// Mitsubishi GX Works2 project: zadatak_1   PLC: FX3S

// task Task_01 (event TRUE, interval 0, priority 31): POU_01

PROGRAM POU_01
VAR
  system_on : BOOL;
  start : BOOL;
  stop_all : BOOL;
  start_all : BOOL;
  fsm_1 : fsm;
  pump_on : BOOL;
  goto_1 : BOOL;
  goto_2 : BOOL;
  goto_3 : BOOL;
  goto_4 : BOOL;
  goto_0 : BOOL;
  cur_state : INT;
  s_0 : BOOL;
  s_1 : BOOL;
  s_2 : BOOL;
  s_3 : BOOL;
  s_4 : BOOL;
  sensor_2 : BOOL;
END_VAR
VAR CONSTANT
  pause : TIME := T#10s;
END_VAR
VAR
  elapsed_time : TIME;
  sensor_1 : BOOL;
  water_rising : BOOL;
  valve_1 : BOOL;
  motor : BOOL;
  water_falling : BOOL;
  valve_2 : BOOL;
  alarm : BOOL;
  TON_1 : TON;
  cnt_cycles_1 : cnt_cycles;
  done : BOOL;
  blink_1 : blink;
  lamp : BOOL;
END_VAR
(* structured ladder/FBD written out as ST: instructions are called as NAME(EN, inputs, outputs); _pN, _eN, _tN stand for wires *)
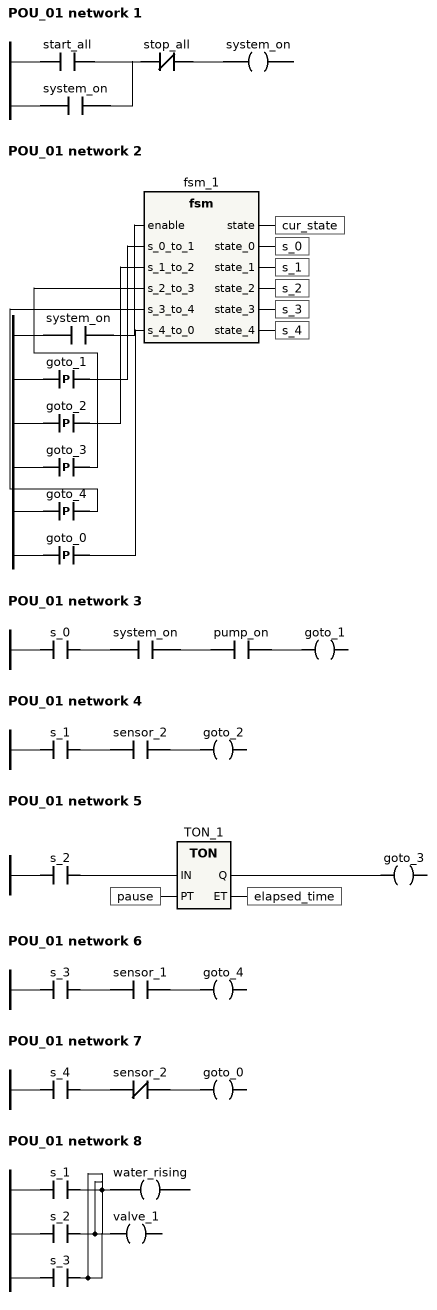
(* network 1 *)
system_on := (start_all OR system_on) AND NOT stop_all;
(* network 2 *)
fsm_1(enable := system_on, s_0_to_1 := LDP(TRUE, goto_1), s_1_to_2 := LDP(TRUE, goto_2), s_2_to_3 := LDP(TRUE, goto_3), s_3_to_4 := LDP(TRUE, goto_4), s_4_to_0 := LDP(TRUE, goto_0), state => cur_state, state_0 => s_0, state_1 => s_1, state_2 => s_2, state_3 => s_3, state_4 => s_4);
(* network 3 *)
goto_1 := s_0 AND system_on AND pump_on;
(* network 4 *)
goto_2 := s_1 AND sensor_2;
(* network 5 *)
TON_1(IN := s_2, PT := pause, ET => elapsed_time);
goto_3 := TON_1.Q;
(* network 6 *)
goto_4 := s_3 AND sensor_1;
(* network 7 *)
goto_0 := s_4 AND NOT sensor_2;
(* network 8 *)
_p1 := s_1 OR s_2 OR s_3;
water_rising := _p1;
valve_1 := _p1;
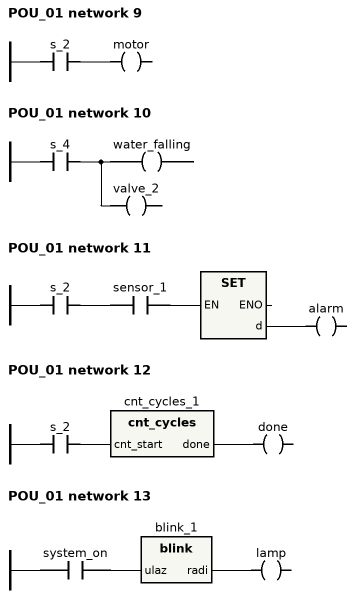
(* network 9 *)
motor := s_2;
(* network 10 *)
water_falling := s_4;
valve_2 := s_4;
(* network 11 *)
SET(s_2 AND sensor_1, _t1);
alarm := _t1;
(* network 12 *)
cnt_cycles_1(cnt_start := s_2);
done := cnt_cycles_1.done;
(* network 13 *)
blink_1(ulaz := system_on);
lamp := blink_1.radi;
END_PROGRAM

FUNCTION_BLOCK fsm
VAR_OUTPUT
  state : INT;
END_VAR
VAR CONSTANT
  cmp_with_0 : INT;
END_VAR
VAR
  is_eqv : ARRAY [0..2] OF BOOL;
END_VAR
VAR_INPUT
  enable : BOOL;
  s_0_to_1 : BOOL;
END_VAR
VAR_OUTPUT
  state_0 : BOOL;
END_VAR
VAR CONSTANT
  cmp_with_1 : INT := 1;
END_VAR
VAR_INPUT
  s_1_to_2 : BOOL;
END_VAR
VAR_OUTPUT
  state_1 : BOOL;
END_VAR
VAR CONSTANT
  cmp_with_2 : INT := 2;
END_VAR
VAR_INPUT
  s_2_to_3 : BOOL;
END_VAR
VAR_OUTPUT
  state_2 : BOOL;
  state_3 : BOOL;
END_VAR
VAR_INPUT
  s_3_to_4 : BOOL;
END_VAR
VAR CONSTANT
  cmp_with_4 : INT := 4;
  cmp_with_3 : INT := 3;
END_VAR
VAR_OUTPUT
  state_4 : BOOL;
END_VAR
VAR_INPUT
  s_4_to_0 : BOOL;
END_VAR
VAR
  blink_1 : blink;
END_VAR
(* structured ladder/FBD written out as ST: instructions are called as NAME(EN, inputs, outputs); _pN, _eN, _tN stand for wires *)
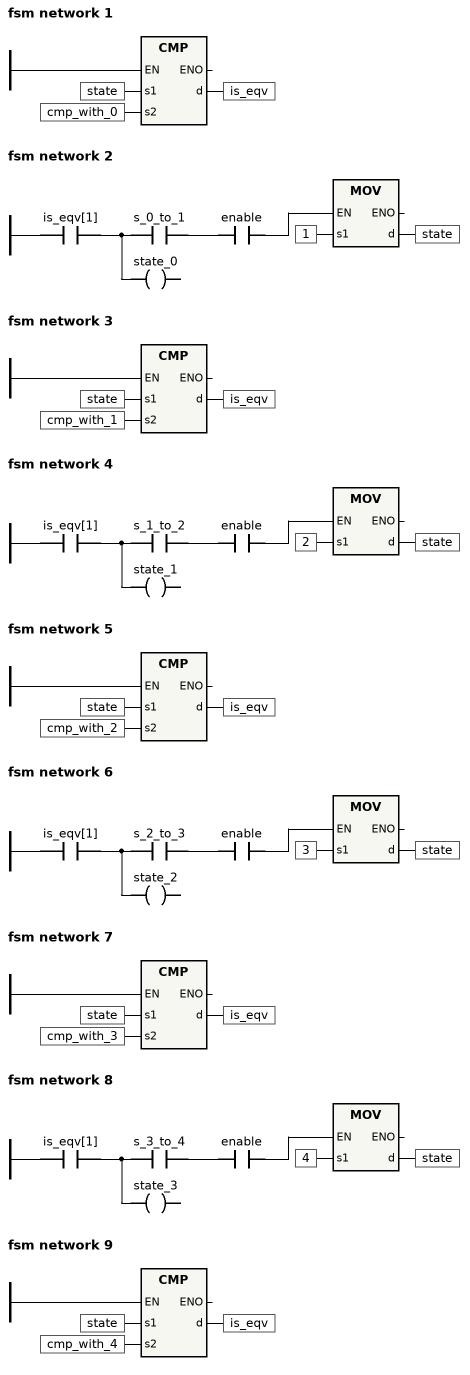
(* network 1 *)
CMP(TRUE, state, cmp_with_0, is_eqv);
(* network 2 *)
MOV(is_eqv[1] AND s_0_to_1 AND enable, 1, state);
state_0 := is_eqv[1];
(* network 3 *)
CMP(TRUE, state, cmp_with_1, is_eqv);
(* network 4 *)
MOV(is_eqv[1] AND s_1_to_2 AND enable, 2, state);
state_1 := is_eqv[1];
(* network 5 *)
CMP(TRUE, state, cmp_with_2, is_eqv);
(* network 6 *)
MOV(is_eqv[1] AND s_2_to_3 AND enable, 3, state);
state_2 := is_eqv[1];
(* network 7 *)
CMP(TRUE, state, cmp_with_3, is_eqv);
(* network 8 *)
MOV(is_eqv[1] AND s_3_to_4 AND enable, 4, state);
state_3 := is_eqv[1];
(* network 9 *)
CMP(TRUE, state, cmp_with_4, is_eqv);
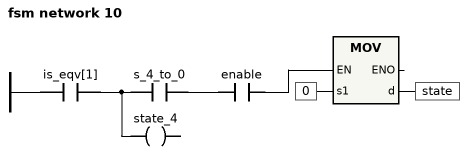
(* network 10 *)
MOV(is_eqv[1] AND s_4_to_0 AND enable, 0, state);
state_4 := is_eqv[1];
END_FUNCTION_BLOCK

FUNCTION_BLOCK cnt_cycles
VAR_INPUT
  cnt_start : BOOL;
END_VAR
VAR
  num_of_cycles : INT;
END_VAR
VAR CONSTANT
  add_1 : INT := 1;
END_VAR
VAR
  is_eqv : ARRAY [0..2] OF BOOL;
END_VAR
VAR CONSTANT
  cmp_with_5 : INT := 5;
END_VAR
VAR_OUTPUT
  done : BOOL;
END_VAR
(* structured ladder/FBD written out as ST: instructions are called as NAME(EN, inputs, outputs); _pN, _eN, _tN stand for wires *)
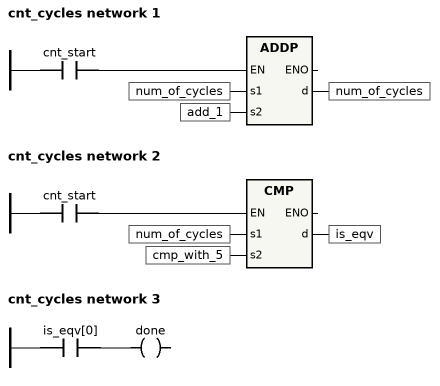
(* network 1 *)
ADDP(cnt_start, num_of_cycles, add_1, num_of_cycles);
(* network 2 *)
CMP(cnt_start, num_of_cycles, cmp_with_5, is_eqv);
(* network 3 *)
done := is_eqv[0];
END_FUNCTION_BLOCK

FUNCTION_BLOCK blink
VAR_INPUT
  ulaz : BOOL;
END_VAR
VAR_OUTPUT
  radi : BOOL;
END_VAR
VAR
  TON_1 : TON;
  TON_2 : TON;
  Tajmer1_izlaz : BOOL;
  Tajmer2_izlaz : BOOL;
  vreme_ton1 : TIME;
  vreme_ton2 : TIME;
END_VAR
IF ulaz=TRUE THEN
	
	TON_1(IN:=NOT Tajmer2_izlaz,PT:= T#1000ms,Q:=Tajmer1_izlaz,ET:=vreme_ton1);
	TON_2(IN:=NOT Tajmer2_izlaz,PT:= T#2000ms,Q:=Tajmer2_izlaz,ET:=vreme_ton2);
	
END_IF;

IF Tajmer1_izlaz=TRUE THEN radi:=TRUE;ELSE radi:=FALSE;
END_IF;
END_FUNCTION_BLOCK
